FUNCTION_BLOCK Write_Influx2 (* Template for a Simple Function Block Type *)
  (* Standard: 61499-1 *)
  (* Version 1.0, 2024-08-01, david *)
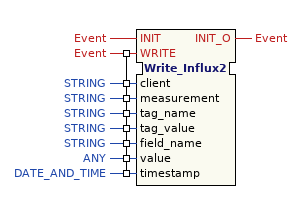
  EVENT_INPUT
    INIT; (* Initialze Function Block *)
    WRITE WITH timestamp, value, field_name, tag_value, tag_name, measurement, client;
  END_EVENT
  EVENT_OUTPUT
    INIT_O; (* Initialze function block confirmation *)
  END_EVENT
  VAR_INPUT
    client : STRING; (* client object *)
    measurement : STRING; (* Name of measurement *)
    tag_name : STRING; (* Name of tag (optional) *)
    tag_value : STRING; (* Value of tag (optional) *)
    field_name : STRING; (* Name of field *)
    value : ANY; (* Field value *)
    timestamp : DATE_AND_TIME; (* timestamp of datapoint (optional) *)
  END_VAR
  ALGORITHM REQ IN ST: (* Normally executed algorithm *)
OUT := IN;
  END_ALGORITHM
END_FUNCTION_BLOCK
